Staubli VAL3: SUB.pjx

--- SUB.pjx ---
Parameters version=s7.5 stackSize=5000 millimeterUnit=true
Program file=delete.pgx
Program file=deleteItem.pgx
Program file=delEvent.pgx
Program file=duplicate.pgx
Program file=find.pgx
Program file=findItem.pgx
Program file=get.pgx
Program file=getItem.pgx
Program file=getProgItem.pgx
Program file=getSize.pgx
Program file=getSizeItem.pgx
Program file=getType.pgx
Program file=insertItem.pgx
Program file=load.pgx
Program file=loadCycle.pgx
Program file=loadPage.pgx
Program file=lookForInstr.pgx
Program file=new.pgx
Program file=onEdit.pgx
Program file=onInsert.pgx
Program file=onProgEnd.pgx
Program file=onRun.pgx
Program file=onStart.pgx
Program file=onStop.pgx
Program file=pasteItem.pgx
Program file=save.pgx
Program file=selectItem.pgx
Program file=setItem.pgx
Program file=showExist.pgx
Program file=unSelectItem.pgx
Data file=SUB.dtx
Library alias=page path=Disk://kernel/template/page/page.pjx
Library alias=use path=Disk://kernel/userPage/userPage.pjx
Library alias=language path=Disk://kernel/language/language.pjx
Library alias=cycleStatus path=Disk://cycleStatus/cycleStatus.pjx
Library alias=saveProg path=Disk://kernel/template/session/saveProg/SUB/SUB.pjx
Library alias=saveData path=Disk://saveData/saveData.pjx
Library alias=instruction path=Disk://../templates/instruction/instruction.pjx
Type name=progItem path=Disk://kernel/template/progItem/progItem.pjx
Type name=InstrItem path=Disk://kernel/template/InstrItem/InstrItem.pjx

--- SUB.dtx ---
num nChar = 89
num nFile = 2
num nPath
public string sItems
string sSession
progItem pEdit
  [0]
    InstrItem iEvent
      [0]
        string sType
        string sData
    string sID
num nKey

--- delete.pgx ---
public program delete(string x_sName, num x_nResult)
  local string l_sItem
  local num l_nDefault
begin
  //
  // delete the select program in
  //
  if isDefined(saveProg:pProg[x_sName])
    // delete
    delete(saveProg:pProg[x_sName])
  endIf
end

--- deleteItem.pgx ---
public program deleteItem(num x_nIndex, num& x_nResult[])
  local num l_nFound
  local num l_nSize
  local num i
  local InstrItem l_sEvent
begin
  //
  // delete the selected field
  //
  call getSizeItem(l_nSize)
  l_nFound=0
  for i=0 to (l_nSize-1)
    call getItem(l_sEvent,i)
    if find(l_sEvent.sType,"#")!=-1
      l_nFound=-1
      call delEvent(i)
      i=i-1
    endIf
  endFor
  //
  // if there are no marked events delete the select one
  //
  if x_nIndex!=-1 and l_nFound==0
    call delEvent(x_nIndex)
  endIf
end

--- delEvent.pgx ---
program delEvent(num x_nIndex)
begin
  // delete the item
  if size(pEdit.iEvent)>1
    delete(pEdit.iEvent[x_nIndex])
  else
    pEdit.iEvent.sType=""
    pEdit.iEvent.sData=""
  endIf
end

--- duplicate.pgx ---
public program duplicate(string x_sCopy, string x_sPaste, num& x_nResult[])
  local num i
  local num l_nSize
  local string l_sItem
  local bool l_bFound
begin
  //
  // return -1 if present
  //
  // create a new one
  call new(x_sPaste,i)
  // duplicate
  saveProg:pProg[x_sPaste]=saveProg:pProg[x_sCopy]
  saveProg:pProg[x_sPaste].sID=x_sPaste
end

--- find.pgx ---
public program find(string& x_sItem[], bool& x_bFound[])
  local num i
  local num l_nSize
  local string l_sEvent
begin
  // search a  SUB program
  // check if the item has been found
  x_bFound=isDefined(saveProg:pProg[x_sItem])
end

--- findItem.pgx ---
public program findItem(InstrItem x_iItem, num& x_nResult[], bool x_bUseSession)
// procedure
  local num i
  local num j
  local num l_nSize
  local string l_sProgName
  local bool l_bFound
  local num l_nSizeItem
  local InstrItem l_iItem
  local num z
  local string l_sSession
  local string l_sMessage
begin
  //
  // search in all of the program the x_iItem
  //
  call getSize(l_nSize)
  for i=0 to (l_nSize-1)
    // load all the program
    call get(l_sProgName,i)
    if l_sProgName!=""
      // SHOW THE program name
      call saveData:getSession(l_sSession)
      l_sMessage="SESSION:"+l_sSession+">SUB "+l_sProgName
      call use:typeLen(1,5,l_sMessage,38)
      // load the select program and search inside
      call load(l_sProgName,x_nResult)
      if x_nResult==0
        // SEARCH IN ALL THE ITEMS
        call getSizeItem(l_nSizeItem)
        if l_nSize!=0
          for j=0 to (l_nSizeItem-1)
            call getItem(l_iItem,j)
            // look inside
            l_bFound=(l_iItem.sType==x_iItem.sType and(l_iItem.sData==x_iItem.sData or find(l_iItem.sData," "+x_iItem.sData)!=-1))
            // use nested items
            if x_iItem.sType=="IN" or x_iItem.sType=="OUT" or x_iItem.sType=="NUM"
              l_bFound=l_bFound or (find(l_iItem.sData,x_iItem.sType)!=-1 and find(l_iItem.sData," "+x_iItem.sData)!=-1)
            else
              l_bFound=l_bFound or (find(l_iItem.sData,x_iItem.sType)!=-1 and find(l_iItem.sData+"#"," "+x_iItem.sData+"#")!=-1)
            endIf
            // FOUND IT
            if l_bFound
              x_nResult=-1
              call language:message(l_sMessage,23)
              popUpMsg(l_sMessage+x_iItem.sType+" "+x_iItem.sData+chr(10)+"SESSION:"+l_sSession+chr(10)+"SUB: "+l_sProgName+" > "+l_iItem.sType+" "+l_iItem.sData)
              // back
              return
            endIf
          endFor
        endIf
      else
        popUpMsg("error loading...SESSION:"+l_sSession+">SUB "+l_sProgName+" error "+toString("",x_nResult))
      endIf
    endIf
  endFor
end

--- get.pgx ---
public program get(string& x_sItem[], num x_nIndex)
  local string l_sKey
  local num i
begin
  // start from the first
  l_sKey=first(saveProg:pProg)
  // search it
  while l_sKey!=""
    x_sItem=l_sKey
    l_sKey=next(saveProg:pProg[l_sKey])
    if i==x_nIndex
      return
    else
      i=i+1
    endIf
  endWhile
end

--- getItem.pgx ---
public program getItem(InstrItem& x_sItem, num x_nIndex)
begin
  // give back the instruction
  x_sItem=pEdit.iEvent[x_nIndex]
end

--- getProgItem.pgx ---
public program getProgItem(progItem& x_pProgItem, string x_sName)
begin
  if isDefined(saveProg:pProg[x_sName])
    // give back
    x_pProgItem=saveProg:pProg[x_sName]
    x_pProgItem.sID=x_sName
  else

  endIf
end

--- getSize.pgx ---
public program getSize(num& x_nSize[])
  local num i
  local num l_nSize
  local bool l_bFound
  local string l_sEmpty
  local string l_sPath
  local string l_sType
  local string l_sKey
  local string l_sItem
begin
  // give back the size to trajectory field
  x_nSize=size(saveProg:pProg)
end

--- getSizeItem.pgx ---
public program getSizeItem(num& x_nSize[])
begin
  // get the size
  if pEdit.iEvent.sType==""
    x_nSize=0
  else
    x_nSize=size(pEdit.iEvent)
  endIf
end

--- insertItem.pgx ---
public program insertItem(InstrItem& x_sItem[], num x_nIndex)
  local num l_sItem
begin
  if x_nIndex<=0
    x_nIndex=0
  else
    insert(pEdit.iEvent[x_nIndex])
  endIf
  call setItem(x_sItem,x_nIndex)
end

--- load.pgx ---
public program load(string x_sItem, num& x_nResult[])
  local string l_sName
  local string l_sPath
  local string l_sType
  local string l_sMessage
begin
  // check the libPath
  call getType(l_sType)
  // load it
  if find(saveProg:libPath(),saveData:sPathProg)==-1
    l_sPath=saveData:sPathProg+l_sType
    x_nResult=saveProg:libLoad(l_sPath)
    delay(0)
    if saveData:bDebug
      ? "loading SUB..."+l_sPath
    endIf
  endIf
  // reload the edit template
  if isDefined(saveProg:pProg[x_sItem].sID)and x_sItem!=""
    // refresh the iD...
    saveProg:pProg[x_sItem].sID=x_sItem
    // update the select item
    pEdit=saveProg:pProg[x_sItem]
  elseIf x_sItem!=""
    // not FOUND
    call language:message(l_sMessage,-7)
    x_nResult=-1
    popUpMsg(l_sMessage+x_sItem)
    // use an empty one
    pEdit.sID=""
  endIf
end

--- loadCycle.pgx ---
public program loadCycle(string x_sItem, num& x_nResult[])
  local string l_sName
  local string l_sPath
  local string l_sType
begin
  // check the libPath
  call getType(l_sType)
  // load it
  if find(saveProg:libPath(),saveData:sPathProg)==-1
    l_sPath=saveData:sPathProg+l_sType
    x_nResult=saveProg:libLoad(l_sPath)
    if saveData:bDebug
      ? "loading SUB..."+l_sPath
    endIf
  endIf
  // reload the edit template
  if isDefined(saveProg:pProg[x_sItem].sID)and x_sItem!=""
    // refresh the iD...
    saveProg:pProg[x_sItem].sID=x_sItem
    // item found
    x_nResult=0
  endIf
end

--- lookForInstr.pgx ---
program lookForInstr(string& x_sItemToFind[] (dimensions=1), string& x_sItem[] (dimensions=1), bool& x_bFound[] (dimensions=1))
  local num l_nPos
  local bool l_bContinue
begin
  // init
  x_bFound=false
  // look for deep scan or not
  if size(x_sItemToFind)>1
    // find which instruction is
    l_nPos=find(x_sItem,x_sItemToFind)
    if l_nPos!=-1
      // look if the find give a correct answer
      // look before and after
      if l_nPos==0 or (asc(x_sItem,l_nPos-1)<65 or asc(x_sItem,l_nPos-1)>90)
        // continue
        /// OK check for the instruction now
        l_nPos=find(x_sItem,x_sItemToFind[1])
        // look if before is empty
        if asc(x_sItem,l_nPos-1)==32 and l_nPos!=-1
          x_bFound=true
        endIf
      endIf
    endIf
  else
    // NORMAL SEARCH
    if x_sItem==x_sItemToFind
      x_bFound=true
    endIf
  endIf
end

--- new.pgx ---
public program new(string x_sName, num& x_nResult[])
  local string l_sMessage
begin
  // new element
  if insert(saveProg:pProg[x_sName])
    saveProg:pProg[x_sName].sID=x_sName
    x_nResult=0
  else
    call language:message(l_sMessage,-2)
    popUpMsg(l_sMessage)
    x_nResult=-1
  endIf
end

--- onEdit.pgx ---
public program onEdit(string& x_sItem[])
  local num l_nResult
  local num i
  local string l_sItem
  local string l_sType
begin
  //
  // go to the view instruction page
  //
  if size(x_sItem)==1
    // show the items
    if isDefined(saveProg:pProg[x_sItem].iEvent)
      for i=0 to size(saveProg:pProg[x_sItem].iEvent)-1
        l_sItem=l_sItem+saveProg:pProg[x_sItem].iEvent[i].sType+" "+saveProg:pProg[x_sItem].iEvent[i].sData +chr(10)
      endFor
      // remove the last CR
      l_sItem=left(l_sItem,len(l_sItem)-1)
      // show IT
      popUpMsg(l_sItem)
    endIf
  else
    call getType(l_sType)
    saveData:sProgTypeUsing=l_sType
    // load it
    call load(x_sItem,l_nResult)
    // give it back
    x_sItem[1]=x_sItem
    x_sItem="Disk://instruction/PROG/page_instr"
  endIf
end

--- onInsert.pgx ---
public program onInsert(string& x_sItem[])
  local string l_sEvent
  local num i
  local num l_nSize
  local string l_sMessage
  local num l_nKey
  local bool l_bFound
begin
  cls()
  call use:setView(false)
  call use:setSizeList(19,0,19,11)
  //
  // Prog
  //
  call use:listcreate("SUB")
  //
  call getSize(l_nSize)
  // refresh the list
  for i=0 to l_nSize-1
    call get(l_sEvent,i)
    if l_sEvent!=""
      // check it
        call use:listadd(l_sEvent)
    endIf
  endFor
  call use:listupdate(0)
  call language:message(l_sMessage,60)
  call use:typeLen(0,13,l_sMessage,40)
  do
    l_nKey=get()
    call use:listevent(l_nKey,i,x_sItem)
  until l_nKey==270 or l_nKey==255
  if l_nKey==255
    x_sItem=""
  endIf
end

--- onRun.pgx ---
public program onRun(string& x_sItem[])
  local num i
  local string l_sEvent
  local num l_nId
  local num l_nOffset
  local num l_nMoveId
  local bool l_bToStop
  local InstrItem l_iInstr
  local string l_sPath
  local num l_nResult
  local progItem l_pProgItem
  local num l_nIdEvent
begin
  // save the last item..
  l_nIdEvent=cycleStatus:nEvent
  l_pProgItem=cycleStatus:pCycleProg
  // PROG NAME x_sItem
  call loadCycle(x_sItem,l_nResult)
  // continue
  if l_nResult==0
    // SET THE CALL SUB..
    if isDefined(saveProg:pProg[x_sItem])
      saveProg:pProg[x_sItem].sID="SUB "+x_sItem
      l_nOffset=0
      call cycleStatus:getLastId(l_nMoveId)
      // print to screen define the pCycleProg
      cycleStatus:pCycleProg=saveProg:pProg[x_sItem]
      // execute all the action...
      for i=0 to size(saveProg:pProg[x_sItem].iEvent)-1
        l_iInstr=saveProg:pProg[x_sItem].iEvent[i]
        //
        // INSTRUCTION
        //
        if l_iInstr.sType!=""
          //refresh the cycleStatus
          l_sEvent=l_iInstr.sType+" "+l_iInstr.sData
          ? "ACTION RUNNING,"+l_sEvent+",ID="+toString(".3",getMoveId())+","+toString(".3",clock()-cycleStatus:nTime)+",MoveID="+toString("",l_nMoveId)+",Dist="+toString(".2",l_nOffset)
          call cycleStatus:printLog("  -"+l_sEvent)
          cycleStatus:sToShow=l_sEvent
          cycleStatus:sLastAction=l_sEvent
          cycleStatus:nEvent=i
          //
          // RUN THE ACTION
          //
          call saveData:getPathInstr(l_iInstr.sType,l_sPath)
          instruction:libLoad(l_sPath)
          delay(0)
          call instruction:onRun(l_iInstr.sData)
        else
          l_bToStop=true
        endIf
      endFor
      // reinizialize
      cycleStatus:nEvent=l_nIdEvent
      cycleStatus:pCycleProg=l_pProgItem
      use:bUseRefresh=true
    else
      l_bToStop=true
    endIf
  else
    l_bToStop=true
  endIf
  // check the error...
  if l_bToStop
    // error message
    popUpMsg("SUB not FOUND")
    cycleStatus:bToStop=true
    watch(cycleStatus:bToStop==false,1)
  endIf
end

--- onStart.pgx ---
public program onStart(string& x_sItem[])
  local string l_sType
  local num i
  local string l_sPath
  local num l_nResult
  local string l_sName
begin
  // on Start

end

--- onStop.pgx ---
public program onStop(string& x_sItem[] (dimensions=1))
begin
end

--- pasteItem.pgx ---
public program pasteItem(num& x_nIndex[])
  local num l_nSize
  local num i
  local InstrItem l_sItem
  local num l_nTemp
  local string l_sRight
begin
  call getSizeItem(l_nSize)
  l_nTemp=x_nIndex+1
  for i=0 to (l_nSize-1)
    call getItem(l_sItem,i)
    if find(l_sItem.sType,"#")!=-1
      if l_nTemp<=i
        i=i+1
      endIf
      l_sItem.sType=right(l_sItem.sType,len(l_sItem.sType)-1)
      call insertItem(l_sItem,l_nTemp)
      l_nTemp=l_nTemp+1
      l_nSize=l_nSize+1
    endIf
  endFor
  // unselect all
  call unSelectItem()
end

--- save.pgx ---
public program save(string x_sName, num& x_nResult[])
begin
  // save it
  if isDefined(saveProg:pProg[x_sName]) and pEdit.iEvent.sType!=""
    saveProg:pProg[x_sName]=pEdit
  endIf
  x_nResult=saveProg:libSave()
end

--- selectItem.pgx ---
public program selectItem(num x_nIndex)
  local InstrItem l_sItem
begin
  //
  // select or unselect one item
  //
  call getItem(l_sItem,x_nIndex)
  if find(l_sItem.sType,"#")==-1
    l_sItem.sType="#"+l_sItem.sType
  else
    l_sItem.sType=right(l_sItem.sType,len(l_sItem.sType)-1)
  endIf
  // set Item
  call setItem(l_sItem,x_nIndex)
end

--- setItem.pgx ---
public program setItem(InstrItem& x_sItem[], num& x_nIndex[])
begin
  // set IT
  pEdit.iEvent[x_nIndex]=x_sItem
end

--- unSelectItem.pgx ---
public program unSelectItem()
  local InstrItem l_sEvent
  local num i
  local num l_nSize
begin
  // deselect all
  call getSizeItem(l_nSize)
  for i=0 to (l_nSize-1)
    call getItem(l_sEvent,i)
    if find(l_sEvent.sType,"#")!=-1
      l_sEvent.sType=right(l_sEvent.sType,len(l_sEvent.sType)-1)
      call setItem(l_sEvent,i)
    endIf
  endFor
end
